(* Logix 5000 project; controller Comas_L4 vendor 1 type 14 code 193 rev 30.11; software revision 30.02; part 8 of 12 *)
(* tags used below, declared in another part *)
   AOI_Pilotage_Codeur_Vitesse_Moy : Pilotage_Vitesse_Rapide_V4;
   Axe_Codeur_Four : AXIS_CIP_DRIVE;
   Axe_Coupe_Fil : AXIS_CIP_DRIVE;
   Axe_Horizontal_Droit : AXIS_CIP_DRIVE;
   Axe_Horizontal_Gauche : AXIS_CIP_DRIVE;
   Axe_Pompe_Doseuse : AXIS_CIP_DRIVE;
   Axe_Rouleaux_Canneles : AXIS_CIP_DRIVE;
   Axe_Vertical_Droit : AXIS_CIP_DRIVE;
   Axe_Vertical_Gauche : AXIS_CIP_DRIVE;
   Axe_Virtuel_Codeur : AXIS_VIRTUAL;
   Axe_Virtuel_Maitre : AXIS_VIRTUAL;
   CamGenerator_Coupe_Fil : AOI_CamGenerator_ST;
   CamGenerator_Horizontal : AOI_CamGenerator_ST;
   CamGenerator_Vertical : AOI_CamGenerator_ST;
   CO_Acquit_defaut : BOOL;
   CO_Axe_Codeur_Four_Conv_Cons : REAL;
   CO_Axe_Codeur_Four_OK : BOOL;
   CO_Axe_Codeur_Four_PosUnwind : DINT;
   CO_Axe_Coupe_Fil_Conv_Cons : REAL;
   CO_Axe_Coupe_Fil_OK : BOOL;
   CO_Axe_Coupe_Fil_PosUnwind : DINT;
   CO_Axe_Horizontal_Droit_OK : BOOL;
   CO_Axe_Horizontal_Gauche_OK : BOOL;
   CO_Axe_Pompe_Doseuse_OK : BOOL;
   CO_Axe_Rouleaux_Canneles_OK : BOOL;
   CO_Axe_Vertical_Droit_OK : BOOL;
   CO_Axe_Vertical_Gauche_OK : BOOL;
   CO_Axe_Virtuel_Codeur_Conv_Cons : REAL;
   CO_Axe_Virtuel_Codeur_PosUnwind : DINT;
   CO_Axe_Virtuel_Maitre_Conv_Cons : REAL;
   CO_Axe_Virtuel_Maitre_PosUnwind : DINT;
   CO_BP_Coupe_Fil_Neg : BOOL;
   CO_BP_Coupe_Fil_Pos : BOOL;
   CO_BP_Horizontal_Droit_Neg : BOOL;
   CO_BP_Horizontal_Droit_Pos : BOOL;
   CO_BP_Horizontal_Gauche_Neg : BOOL;
   CO_BP_Horizontal_Gauche_Pos : BOOL;
   CO_BP_Pompe_Doseuse_Neg : BOOL;
   CO_BP_Pompe_Doseuse_Pos : BOOL;
   CO_BP_Rouleaux_Canneles_Neg : BOOL;
   CO_BP_Rouleaux_Canneles_Pos : BOOL;
   CO_BP_Vertical_Droit_Neg : BOOL;
   CO_BP_Vertical_Droit_Pos : BOOL;
   CO_BP_Vertical_Gauche_Neg : BOOL;
   CO_BP_Vertical_Gauche_Pos : BOOL;
   CO_Defaut_CamGenerator_Coupe_Fil : BOOL;
   CO_Defaut_CamGenerator_Horizontal : BOOL;
   CO_Defaut_CamGenerator_Vertical : BOOL;
   CO_Defaut_Eth_Codeur_Four : BOOL;
   CO_Defaut_Eth_Var_Coupe_Fil : BOOL;
   CO_Defaut_Eth_Var_H_Droit : BOOL;
   CO_Defaut_Eth_Var_H_Gauche : BOOL;
   CO_Defaut_Eth_Var_Pompe_Doseuse : BOOL;
   CO_Defaut_Eth_Var_Rouleaux : BOOL;
   CO_Defaut_Eth_Var_V_Droit : BOOL;
   CO_Defaut_Eth_Var_V_Gauche : BOOL;
   CO_Defaut_FDC_Amont_Horizontal_Droit : BOOL;
   CO_Defaut_FDC_Amont_Horizontal_Gauche : BOOL;
   CO_Defaut_FDC_Aval_Horizontal_Droit : BOOL;
   CO_Defaut_FDC_Aval_Horizontal_Gauche : BOOL;
   CO_Defaut_FDC_Bas_Vertical_Droit : BOOL;
   CO_Defaut_FDC_Bas_Vertical_Gauche : BOOL;
   CO_Defaut_FDC_Coupe_Fil_Droit : BOOL;
   CO_Defaut_FDC_Coupe_Fil_Gauche : BOOL;
   CO_Defaut_FDC_Haut_Vertical_Droit : BOOL;
   CO_Defaut_FDC_Haut_Vertical_Gauche : BOOL;
   CO_Defaut_Presence_Coupe_Fil : BOOL;
   CO_en_Marche : BOOL;
   CO_Machine_sans_defaut : BOOL;
   CO_Messages_En : STRING[380];
   CO_Raz_Axe : BOOL;
   CO_Temp_Vitesse_Four : REAL;
   Consigne_Acc_Decc_Manu_Degre : DINT;
   Consigne_Vitesse_Manu_Degre_Seconde : REAL;
   Consigne_Vitesse_Manu_Tour_Seconde : REAL;
   ENT_CO_Presence_Coupe_Fil : ALIAS FOR Local:2:I.Pt00.Data;
   L_Ms_Index_Codeur_Four : DINT;
   L_Ms_Index_Coupe_Fil : DINT;
   L_Ms_Index_H_Droit : DINT;
   L_Ms_Index_H_Gauche : DINT;
   L_Ms_Index_Pompe_Doseuse : DINT;
   L_Ms_Index_Rouleaux : DINT;
   L_Ms_Index_V_Droit : DINT;
   L_Ms_Index_V_Gauche : DINT;
   Message_Axe_Codeur_Four : Message_Axe;
   Message_Axe_Coupe_Fil : Message_Axe;
   Message_Axe_H_Droit : Message_Axe;
   Message_Axe_H_Gauche : Message_Axe;
   Message_Axe_Pompe_Doseuse : Message_Axe;
   Message_Axe_Rouleaux : Message_Axe;
   Message_Axe_V_Droit : Message_Axe;
   Message_Axe_V_Gauche : Message_Axe;
   Message_Defaut_Codeur_Four : STRING;
   Message_Defaut_Coupe_Fil : STRING;
   Message_Defaut_H_Droit : STRING;
   Message_Defaut_H_Gauche : STRING;
   Message_Defaut_Pompe_Doseuse : STRING;
   Message_Defaut_Rouleaux : STRING;
   Message_Defaut_V_Droit : STRING;
   Message_Defaut_V_Gauche : STRING;
   Raz_Axe_Coupe_Fil : Raz_Axe;
   Raz_Axe_H_Droit : Raz_Axe;
   Raz_Axe_H_Gauche : Raz_Axe;
   Raz_Axe_Pompe_Doseuse : Raz_Axe;
   Raz_Axe_Rouleaux : Raz_Axe;
   Raz_Axe_V_Droit : Raz_Axe;
   Raz_Axe_V_Gauche : Raz_Axe;
   RECETTE_EC : UDT_RECIPE;
   RSW_CO_Activation_Nettoyage : BOOL;
   RSW_CO_BP_Coupe_Fil_Neg : BOOL;
   RSW_CO_BP_Coupe_Fil_Pos : BOOL;
   RSW_CO_BP_Horizontal_Droit_Neg : BOOL;
   RSW_CO_BP_Horizontal_Droit_Pos : BOOL;
   RSW_CO_BP_Horizontal_Gauche_Neg : BOOL;
   RSW_CO_BP_Horizontal_Gauche_Pos : BOOL;
   RSW_CO_BP_Horizontal_Neg : BOOL;
   RSW_CO_BP_Horizontal_Pos : BOOL;
   RSW_CO_BP_Pompe_Doseuse_Neg : BOOL;
   RSW_CO_BP_Pompe_Doseuse_Pos : BOOL;
   RSW_CO_BP_Rouleaux_Canneles_Neg : BOOL;
   RSW_CO_BP_Rouleaux_Canneles_Pos : BOOL;
   RSW_CO_BP_Vertical_Droit_Neg : BOOL;
   RSW_CO_BP_Vertical_Droit_Pos : BOOL;
   RSW_CO_BP_Vertical_Gauche_Neg : BOOL;
   RSW_CO_BP_Vertical_Gauche_Pos : BOOL;
   RSW_CO_BP_Vertical_Neg : BOOL;
   RSW_CO_BP_Vertical_Pos : BOOL;
   RSW_CO_NB_Rangs_minutes : REAL;
   Test_Coupe_Fil : Test_Axe_Avec_Autorisation;
   Test_Coupe_Fil_EN : BOOL;
   Test_Horizontal_Droit : Test_Axe_Avec_Autorisation;
   Test_Horizontal_Droit_EN : BOOL;
   Test_Horizontal_Gauche : Test_Axe_Avec_Autorisation;
   Test_Horizontal_Gauche_EN : BOOL;
   Test_Pompe_Doseuse : Test_Axe_Avec_Autorisation;
   Test_Pompe_Doseuse_EN : BOOL;
   Test_Rouleaux_Canneles : Test_Axe_Avec_Autorisation;
   Test_Rouleaux_Canneles_EN : BOOL;
   Test_Vertical_Droit : Test_Axe_Avec_Autorisation;
   Test_Vertical_Droit_EN : BOOL;
   Test_Vertical_Gauche : Test_Axe_Avec_Autorisation;
   Test_Vertical_Gauche_EN : BOOL;
   Vitesse_Moy_Codeur : REAL;

PROGRAM Comas   (* main routine A00_Appel *)

ROUTINE A00_Appel   (* ladder *)
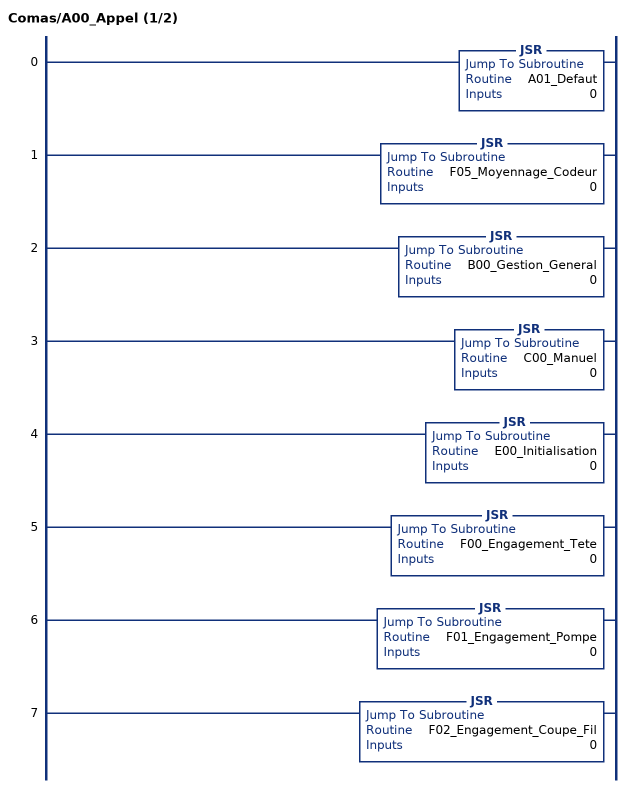
   0: JSR(A01_Defaut,0);
   1: JSR(F05_Moyennage_Codeur,0);
   2: JSR(B00_Gestion_General,0);
   3: JSR(C00_Manuel,0);
   4: JSR(E00_Initialisation,0);
   5: JSR(F00_Engagement_Tete,0);
   6: JSR(F01_Engagement_Pompe,0);
   7: JSR(F02_Engagement_Coupe_Fil,0);
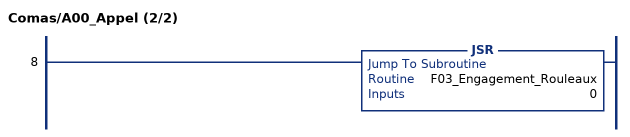
   8: JSR(F03_Engagement_Rouleaux,0);
END_ROUTINE

ROUTINE A01_Defaut   (* ladder *)
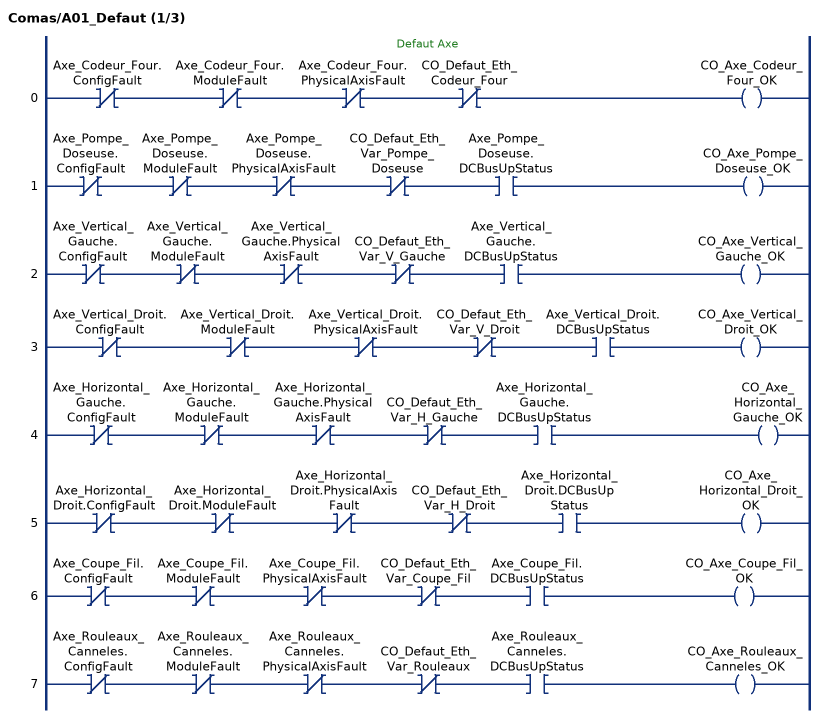
   // Defaut Axe
   0: XIO(Axe_Codeur_Four.ConfigFault)XIO(Axe_Codeur_Four.ModuleFault)XIO(Axe_Codeur_Four.PhysicalAxisFault)XIO(CO_Defaut_Eth_Codeur_Four)OTE(CO_Axe_Codeur_Four_OK);
   1: XIO(Axe_Pompe_Doseuse.ConfigFault)XIO(Axe_Pompe_Doseuse.ModuleFault)XIO(Axe_Pompe_Doseuse.PhysicalAxisFault)XIO(CO_Defaut_Eth_Var_Pompe_Doseuse)XIC(Axe_Pompe_Doseuse.DCBusUpStatus)OTE(CO_Axe_Pompe_Doseuse_OK);
   2: XIO(Axe_Vertical_Gauche.ConfigFault)XIO(Axe_Vertical_Gauche.ModuleFault)XIO(Axe_Vertical_Gauche.PhysicalAxisFault)XIO(CO_Defaut_Eth_Var_V_Gauche)XIC(Axe_Vertical_Gauche.DCBusUpStatus)OTE(CO_Axe_Vertical_Gauche_OK);
   3: XIO(Axe_Vertical_Droit.ConfigFault)XIO(Axe_Vertical_Droit.ModuleFault)XIO(Axe_Vertical_Droit.PhysicalAxisFault)XIO(CO_Defaut_Eth_Var_V_Droit)XIC(Axe_Vertical_Droit.DCBusUpStatus)OTE(CO_Axe_Vertical_Droit_OK);
   4: XIO(Axe_Horizontal_Gauche.ConfigFault)XIO(Axe_Horizontal_Gauche.ModuleFault)XIO(Axe_Horizontal_Gauche.PhysicalAxisFault)XIO(CO_Defaut_Eth_Var_H_Gauche)XIC(Axe_Horizontal_Gauche.DCBusUpStatus)OTE(CO_Axe_Horizontal_Gauche_OK);
   5: XIO(Axe_Horizontal_Droit.ConfigFault)XIO(Axe_Horizontal_Droit.ModuleFault)XIO(Axe_Horizontal_Droit.PhysicalAxisFault)XIO(CO_Defaut_Eth_Var_H_Droit)XIC(Axe_Horizontal_Droit.DCBusUpStatus)OTE(CO_Axe_Horizontal_Droit_OK);
   6: XIO(Axe_Coupe_Fil.ConfigFault)XIO(Axe_Coupe_Fil.ModuleFault)XIO(Axe_Coupe_Fil.PhysicalAxisFault)XIO(CO_Defaut_Eth_Var_Coupe_Fil)XIC(Axe_Coupe_Fil.DCBusUpStatus)OTE(CO_Axe_Coupe_Fil_OK);
   7: XIO(Axe_Rouleaux_Canneles.ConfigFault)XIO(Axe_Rouleaux_Canneles.ModuleFault)XIO(Axe_Rouleaux_Canneles.PhysicalAxisFault)XIO(CO_Defaut_Eth_Var_Rouleaux)XIC(Axe_Rouleaux_Canneles.DCBusUpStatus)OTE(CO_Axe_Rouleaux_Canneles_OK);
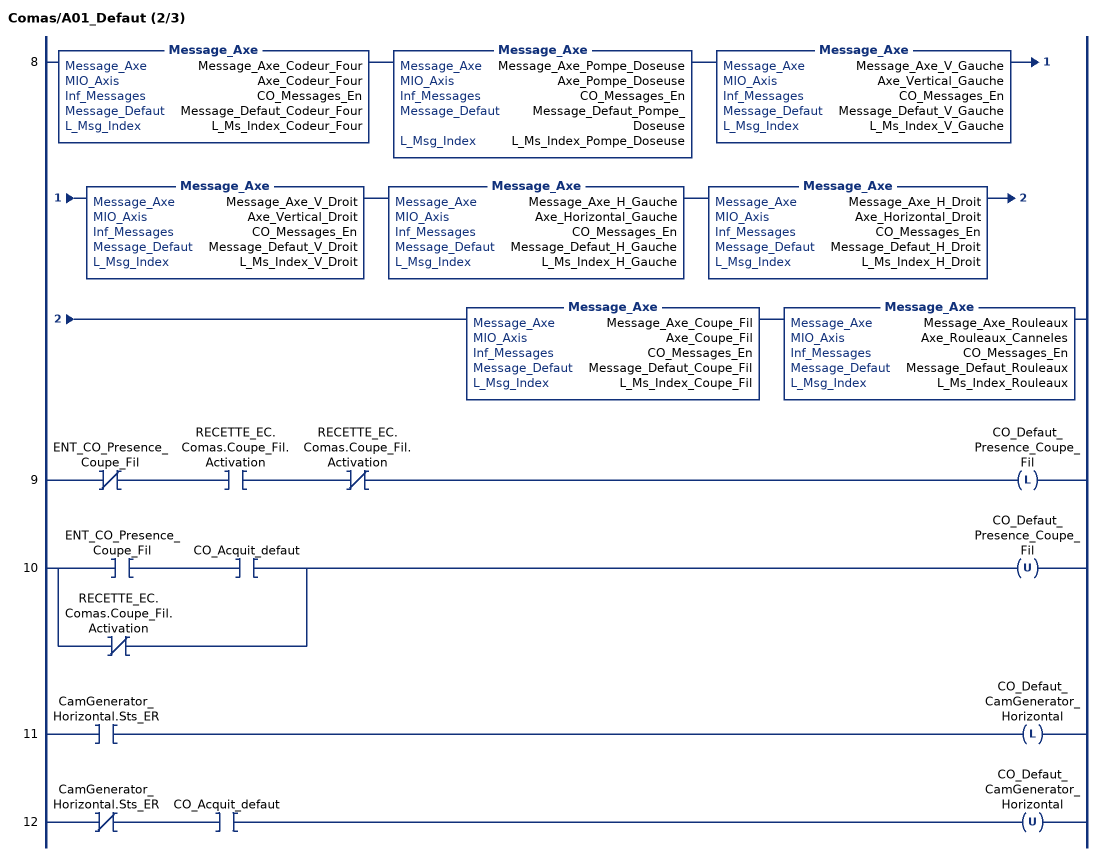
   8: Message_Axe(Message_Axe_Codeur_Four,Axe_Codeur_Four,CO_Messages_En,Message_Defaut_Codeur_Four,L_Ms_Index_Codeur_Four)Message_Axe(Message_Axe_Pompe_Doseuse,Axe_Pompe_Doseuse,CO_Messages_En,Message_Defaut_Pompe_Doseuse,L_Ms_Index_Pompe_Doseuse)Message_Axe(Message_Axe_V_Gauche,Axe_Vertical_Gauche,CO_Messages_En,Message_Defaut_V_Gauche,L_Ms_Index_V_Gauche)Message_Axe(Message_Axe_V_Droit,Axe_Vertical_Droit,CO_Messages_En,Message_Defaut_V_Droit,L_Ms_Index_V_Droit)Message_Axe(Message_Axe_H_Gauche,Axe_Horizontal_Gauche,CO_Messages_En,Message_Defaut_H_Gauche,L_Ms_Index_H_Gauche)Message_Axe(Message_Axe_H_Droit,Axe_Horizontal_Droit,CO_Messages_En,Message_Defaut_H_Droit,L_Ms_Index_H_Droit)Message_Axe(Message_Axe_Coupe_Fil,Axe_Coupe_Fil,CO_Messages_En,Message_Defaut_Coupe_Fil,L_Ms_Index_Coupe_Fil)Message_Axe(Message_Axe_Rouleaux,Axe_Rouleaux_Canneles,CO_Messages_En,Message_Defaut_Rouleaux,L_Ms_Index_Rouleaux);
   9: XIO(ENT_CO_Presence_Coupe_Fil)XIC(RECETTE_EC.Comas.Coupe_Fil.Activation)XIO(RECETTE_EC.Comas.Coupe_Fil.Activation)OTL(CO_Defaut_Presence_Coupe_Fil);
   10: [XIC(ENT_CO_Presence_Coupe_Fil) XIC(CO_Acquit_defaut) ,XIO(RECETTE_EC.Comas.Coupe_Fil.Activation) ]OTU(CO_Defaut_Presence_Coupe_Fil);
   11: XIC(CamGenerator_Horizontal.Sts_ER)OTL(CO_Defaut_CamGenerator_Horizontal);
   12: XIO(CamGenerator_Horizontal.Sts_ER)XIC(CO_Acquit_defaut)OTU(CO_Defaut_CamGenerator_Horizontal);
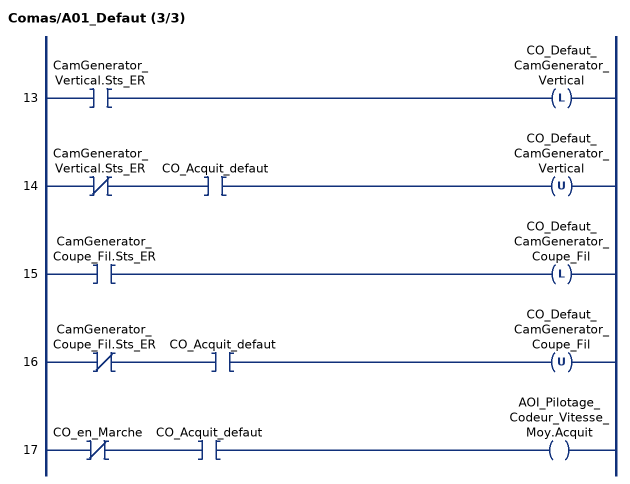
   13: XIC(CamGenerator_Vertical.Sts_ER)OTL(CO_Defaut_CamGenerator_Vertical);
   14: XIO(CamGenerator_Vertical.Sts_ER)XIC(CO_Acquit_defaut)OTU(CO_Defaut_CamGenerator_Vertical);
   15: XIC(CamGenerator_Coupe_Fil.Sts_ER)OTL(CO_Defaut_CamGenerator_Coupe_Fil);
   16: XIO(CamGenerator_Coupe_Fil.Sts_ER)XIC(CO_Acquit_defaut)OTU(CO_Defaut_CamGenerator_Coupe_Fil);
   17: XIO(CO_en_Marche)XIC(CO_Acquit_defaut)OTE(AOI_Pilotage_Codeur_Vitesse_Moy.Acquit);
END_ROUTINE

ROUTINE B00_Gestion_General   (* ladder *)
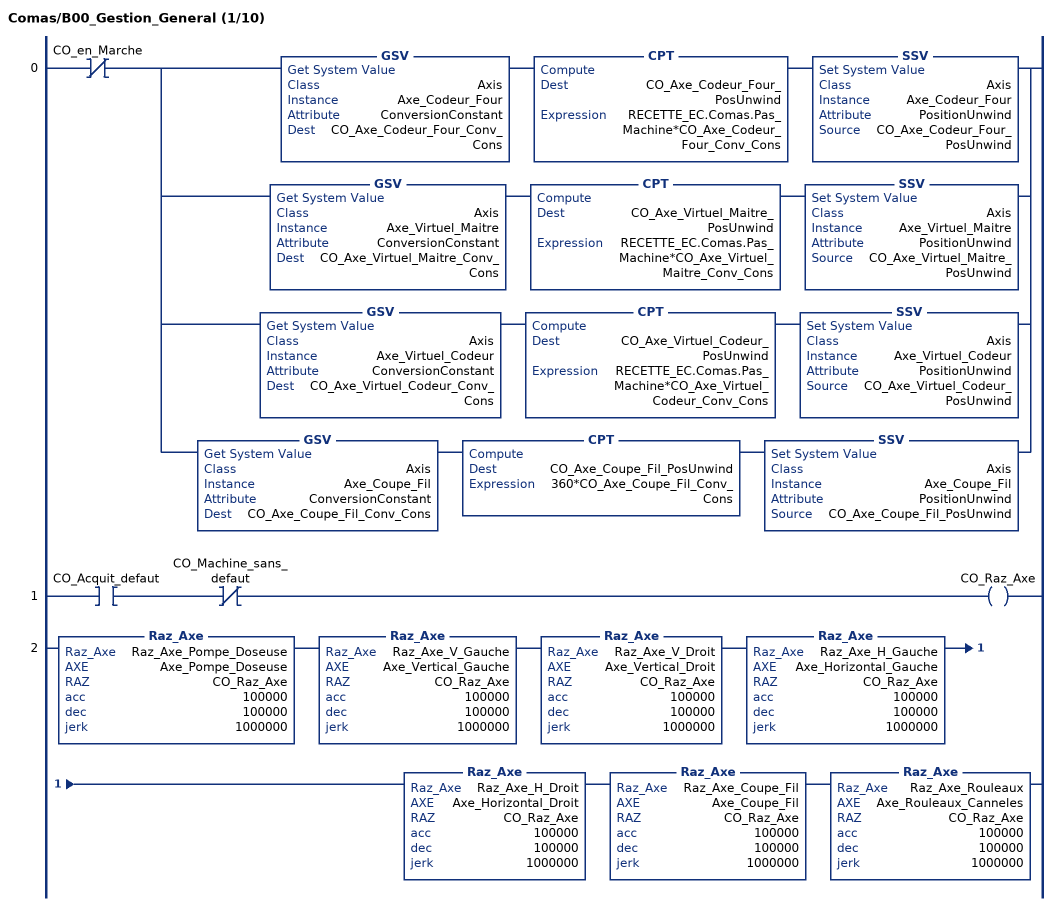
   0: XIO(CO_en_Marche)[GSV(Axis,Axe_Codeur_Four,ConversionConstant,CO_Axe_Codeur_Four_Conv_Cons) CPT(CO_Axe_Codeur_Four_PosUnwind,RECETTE_EC.Comas.Pas_Machine*CO_Axe_Codeur_Four_Conv_Cons) SSV(Axis,Axe_Codeur_Four,PositionUnwind,CO_Axe_Codeur_Four_PosUnwind) ,GSV(Axis,Axe_Virtuel_Maitre,ConversionConstant,CO_Axe_Virtuel_Maitre_Conv_Cons) CPT(CO_Axe_Virtuel_Maitre_PosUnwind,RECETTE_EC.Comas.Pas_Machine*CO_Axe_Virtuel_Maitre_Conv_Cons) SSV(Axis,Axe_Virtuel_Maitre,PositionUnwind,CO_Axe_Virtuel_Maitre_PosUnwind) ,GSV(Axis,Axe_Virtuel_Codeur,ConversionConstant,CO_Axe_Virtuel_Codeur_Conv_Cons) CPT(CO_Axe_Virtuel_Codeur_PosUnwind,RECETTE_EC.Comas.Pas_Machine*CO_Axe_Virtuel_Codeur_Conv_Cons) SSV(Axis,Axe_Virtuel_Codeur,PositionUnwind,CO_Axe_Virtuel_Codeur_PosUnwind) ,GSV(Axis,Axe_Coupe_Fil,ConversionConstant,CO_Axe_Coupe_Fil_Conv_Cons) CPT(CO_Axe_Coupe_Fil_PosUnwind,360*CO_Axe_Coupe_Fil_Conv_Cons) SSV(Axis,Axe_Coupe_Fil,PositionUnwind,CO_Axe_Coupe_Fil_PosUnwind) ];
   1: XIC(CO_Acquit_defaut)XIO(CO_Machine_sans_defaut)OTE(CO_Raz_Axe);
   2: Raz_Axe(Raz_Axe_Pompe_Doseuse,Axe_Pompe_Doseuse,CO_Raz_Axe,100000,100000,1000000)Raz_Axe(Raz_Axe_V_Gauche,Axe_Vertical_Gauche,CO_Raz_Axe,100000,100000,1000000)Raz_Axe(Raz_Axe_V_Droit,Axe_Vertical_Droit,CO_Raz_Axe,100000,100000,1000000)Raz_Axe(Raz_Axe_H_Gauche,Axe_Horizontal_Gauche,CO_Raz_Axe,100000,100000,1000000)Raz_Axe(Raz_Axe_H_Droit,Axe_Horizontal_Droit,CO_Raz_Axe,100000,100000,1000000)Raz_Axe(Raz_Axe_Coupe_Fil,Axe_Coupe_Fil,CO_Raz_Axe,100000,100000,1000000)Raz_Axe(Raz_Axe_Rouleaux,Axe_Rouleaux_Canneles,CO_Raz_Axe,100000,100000,1000000);
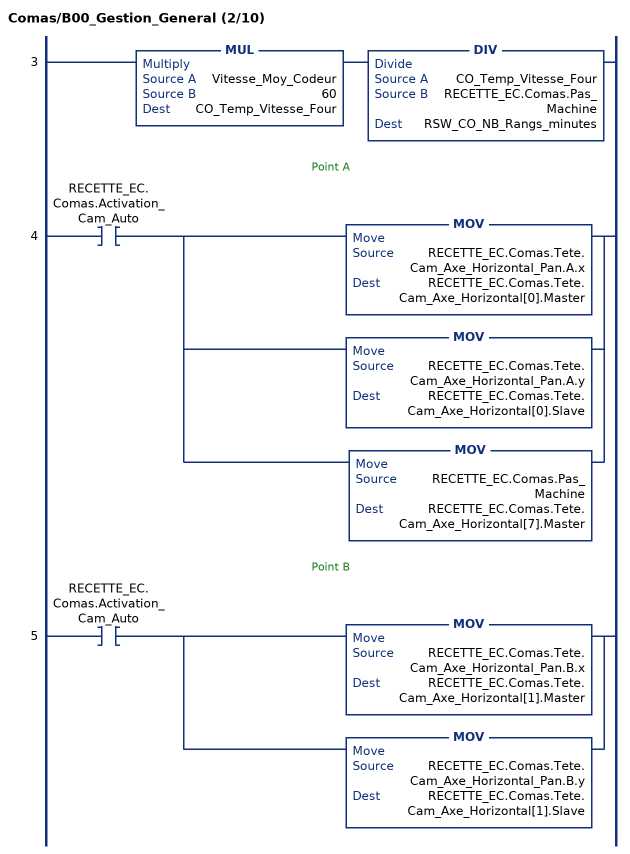
   3: MUL(Vitesse_Moy_Codeur,60,CO_Temp_Vitesse_Four)DIV(CO_Temp_Vitesse_Four,RECETTE_EC.Comas.Pas_Machine,RSW_CO_NB_Rangs_minutes);
   // Point A
   4: XIC(RECETTE_EC.Comas.Activation_Cam_Auto)[MOV(RECETTE_EC.Comas.Tete.Cam_Axe_Horizontal_Pan.A.x,RECETTE_EC.Comas.Tete.Cam_Axe_Horizontal[0].Master) ,MOV(RECETTE_EC.Comas.Tete.Cam_Axe_Horizontal_Pan.A.y,RECETTE_EC.Comas.Tete.Cam_Axe_Horizontal[0].Slave) ,MOV(RECETTE_EC.Comas.Pas_Machine,RECETTE_EC.Comas.Tete.Cam_Axe_Horizontal[7].Master) ];
   // Point B
   5: XIC(RECETTE_EC.Comas.Activation_Cam_Auto)[MOV(RECETTE_EC.Comas.Tete.Cam_Axe_Horizontal_Pan.B.x,RECETTE_EC.Comas.Tete.Cam_Axe_Horizontal[1].Master) ,MOV(RECETTE_EC.Comas.Tete.Cam_Axe_Horizontal_Pan.B.y,RECETTE_EC.Comas.Tete.Cam_Axe_Horizontal[1].Slave) ];
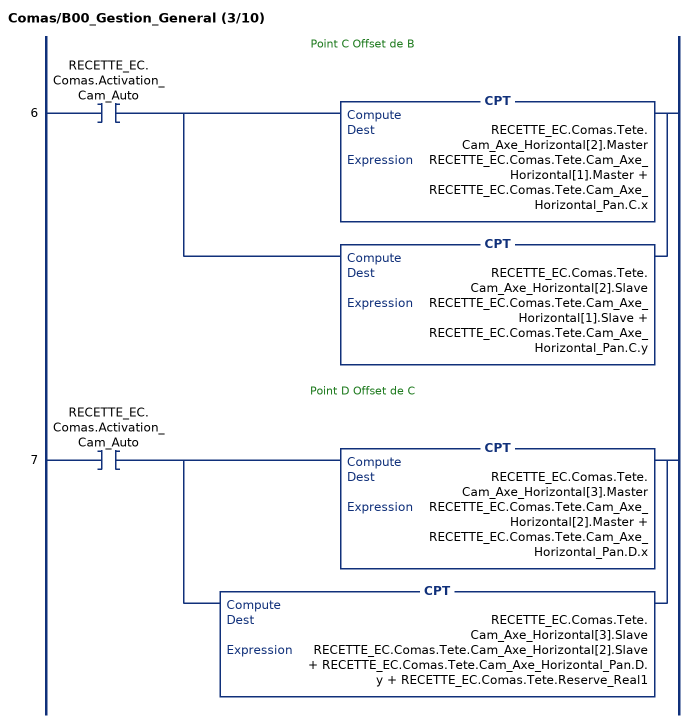
   // Point C Offset de B
   6: XIC(RECETTE_EC.Comas.Activation_Cam_Auto)[CPT(RECETTE_EC.Comas.Tete.Cam_Axe_Horizontal[2].Master,RECETTE_EC.Comas.Tete.Cam_Axe_Horizontal[1].Master + RECETTE_EC.Comas.Tete.Cam_Axe_Horizontal_Pan.C.x) ,CPT(RECETTE_EC.Comas.Tete.Cam_Axe_Horizontal[2].Slave,RECETTE_EC.Comas.Tete.Cam_Axe_Horizontal[1].Slave + RECETTE_EC.Comas.Tete.Cam_Axe_Horizontal_Pan.C.y) ];
   // Point D Offset de C
   7: XIC(RECETTE_EC.Comas.Activation_Cam_Auto)[CPT(RECETTE_EC.Comas.Tete.Cam_Axe_Horizontal[3].Master,RECETTE_EC.Comas.Tete.Cam_Axe_Horizontal[2].Master + RECETTE_EC.Comas.Tete.Cam_Axe_Horizontal_Pan.D.x) ,CPT(RECETTE_EC.Comas.Tete.Cam_Axe_Horizontal[3].Slave,RECETTE_EC.Comas.Tete.Cam_Axe_Horizontal[2].Slave + RECETTE_EC.Comas.Tete.Cam_Axe_Horizontal_Pan.D.y + RECETTE_EC.Comas.Tete.Reserve_Real1) ];
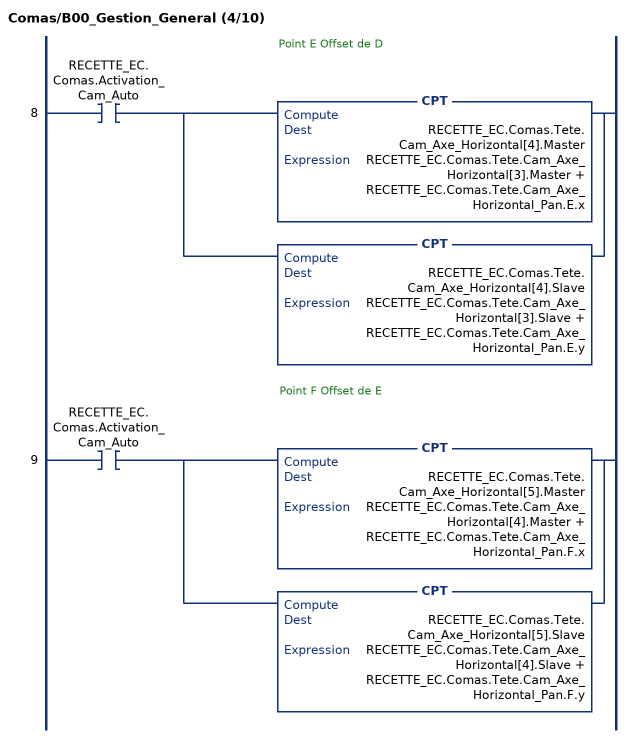
   // Point E Offset de D
   8: XIC(RECETTE_EC.Comas.Activation_Cam_Auto)[CPT(RECETTE_EC.Comas.Tete.Cam_Axe_Horizontal[4].Master,RECETTE_EC.Comas.Tete.Cam_Axe_Horizontal[3].Master + RECETTE_EC.Comas.Tete.Cam_Axe_Horizontal_Pan.E.x) ,CPT(RECETTE_EC.Comas.Tete.Cam_Axe_Horizontal[4].Slave,RECETTE_EC.Comas.Tete.Cam_Axe_Horizontal[3].Slave + RECETTE_EC.Comas.Tete.Cam_Axe_Horizontal_Pan.E.y) ];
   // Point F Offset de E
   9: XIC(RECETTE_EC.Comas.Activation_Cam_Auto)[CPT(RECETTE_EC.Comas.Tete.Cam_Axe_Horizontal[5].Master,RECETTE_EC.Comas.Tete.Cam_Axe_Horizontal[4].Master + RECETTE_EC.Comas.Tete.Cam_Axe_Horizontal_Pan.F.x) ,CPT(RECETTE_EC.Comas.Tete.Cam_Axe_Horizontal[5].Slave,RECETTE_EC.Comas.Tete.Cam_Axe_Horizontal[4].Slave + RECETTE_EC.Comas.Tete.Cam_Axe_Horizontal_Pan.F.y) ];
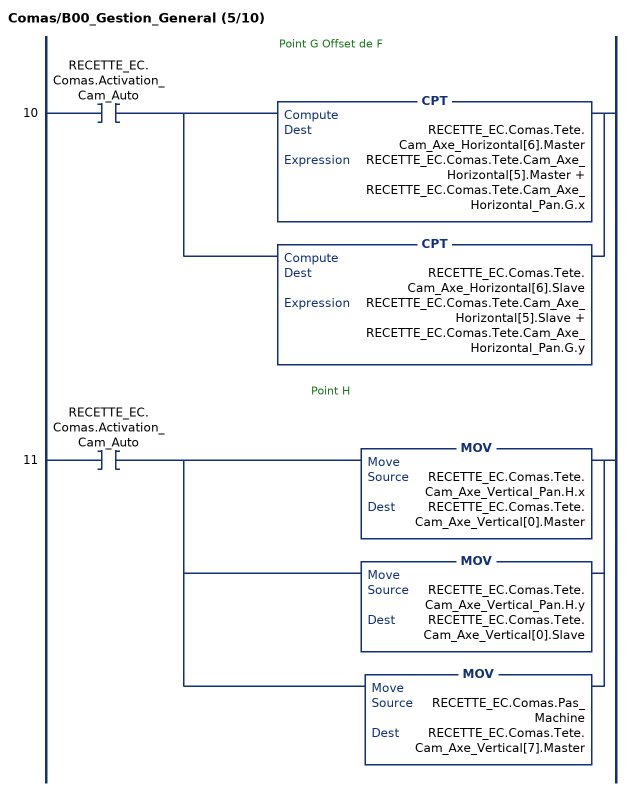
   // Point G Offset de F
   10: XIC(RECETTE_EC.Comas.Activation_Cam_Auto)[CPT(RECETTE_EC.Comas.Tete.Cam_Axe_Horizontal[6].Master,RECETTE_EC.Comas.Tete.Cam_Axe_Horizontal[5].Master + RECETTE_EC.Comas.Tete.Cam_Axe_Horizontal_Pan.G.x) ,CPT(RECETTE_EC.Comas.Tete.Cam_Axe_Horizontal[6].Slave,RECETTE_EC.Comas.Tete.Cam_Axe_Horizontal[5].Slave + RECETTE_EC.Comas.Tete.Cam_Axe_Horizontal_Pan.G.y) ];
   // Point H
   11: XIC(RECETTE_EC.Comas.Activation_Cam_Auto)[MOV(RECETTE_EC.Comas.Tete.Cam_Axe_Vertical_Pan.H.x,RECETTE_EC.Comas.Tete.Cam_Axe_Vertical[0].Master) ,MOV(RECETTE_EC.Comas.Tete.Cam_Axe_Vertical_Pan.H.y,RECETTE_EC.Comas.Tete.Cam_Axe_Vertical[0].Slave) ,MOV(RECETTE_EC.Comas.Pas_Machine,RECETTE_EC.Comas.Tete.Cam_Axe_Vertical[7].Master) ];
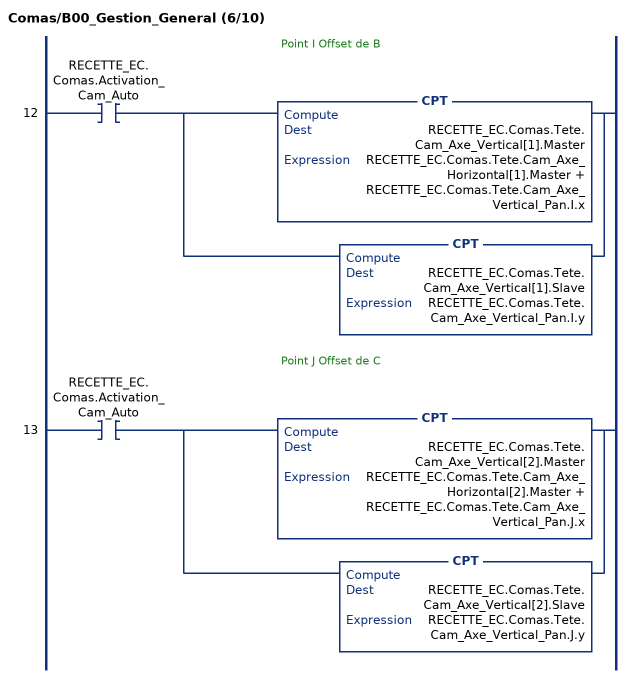
   // Point I Offset de B
   12: XIC(RECETTE_EC.Comas.Activation_Cam_Auto)[CPT(RECETTE_EC.Comas.Tete.Cam_Axe_Vertical[1].Master,RECETTE_EC.Comas.Tete.Cam_Axe_Horizontal[1].Master + RECETTE_EC.Comas.Tete.Cam_Axe_Vertical_Pan.I.x) ,CPT(RECETTE_EC.Comas.Tete.Cam_Axe_Vertical[1].Slave,RECETTE_EC.Comas.Tete.Cam_Axe_Vertical_Pan.I.y) ];
   // Point J Offset de C
   13: XIC(RECETTE_EC.Comas.Activation_Cam_Auto)[CPT(RECETTE_EC.Comas.Tete.Cam_Axe_Vertical[2].Master,RECETTE_EC.Comas.Tete.Cam_Axe_Horizontal[2].Master + RECETTE_EC.Comas.Tete.Cam_Axe_Vertical_Pan.J.x) ,CPT(RECETTE_EC.Comas.Tete.Cam_Axe_Vertical[2].Slave,RECETTE_EC.Comas.Tete.Cam_Axe_Vertical_Pan.J.y) ];
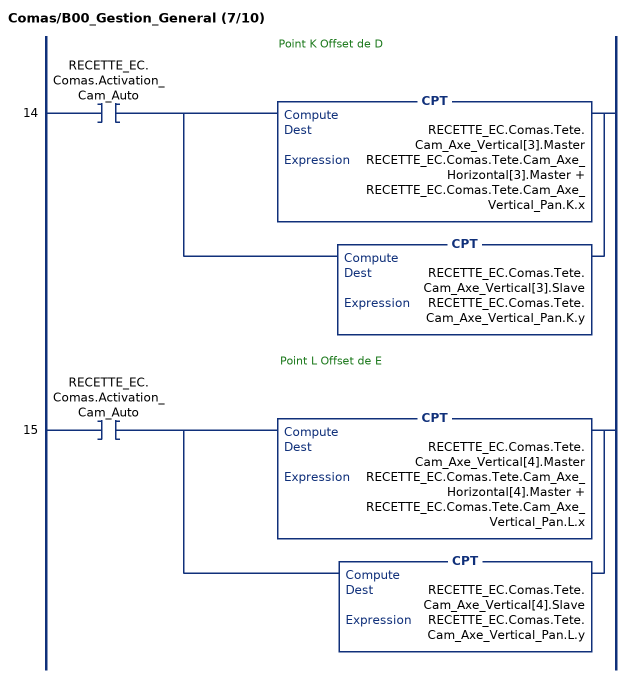
   // Point K Offset de D
   14: XIC(RECETTE_EC.Comas.Activation_Cam_Auto)[CPT(RECETTE_EC.Comas.Tete.Cam_Axe_Vertical[3].Master,RECETTE_EC.Comas.Tete.Cam_Axe_Horizontal[3].Master + RECETTE_EC.Comas.Tete.Cam_Axe_Vertical_Pan.K.x) ,CPT(RECETTE_EC.Comas.Tete.Cam_Axe_Vertical[3].Slave,RECETTE_EC.Comas.Tete.Cam_Axe_Vertical_Pan.K.y) ];
   // Point L Offset de E
   15: XIC(RECETTE_EC.Comas.Activation_Cam_Auto)[CPT(RECETTE_EC.Comas.Tete.Cam_Axe_Vertical[4].Master,RECETTE_EC.Comas.Tete.Cam_Axe_Horizontal[4].Master + RECETTE_EC.Comas.Tete.Cam_Axe_Vertical_Pan.L.x) ,CPT(RECETTE_EC.Comas.Tete.Cam_Axe_Vertical[4].Slave,RECETTE_EC.Comas.Tete.Cam_Axe_Vertical_Pan.L.y) ];
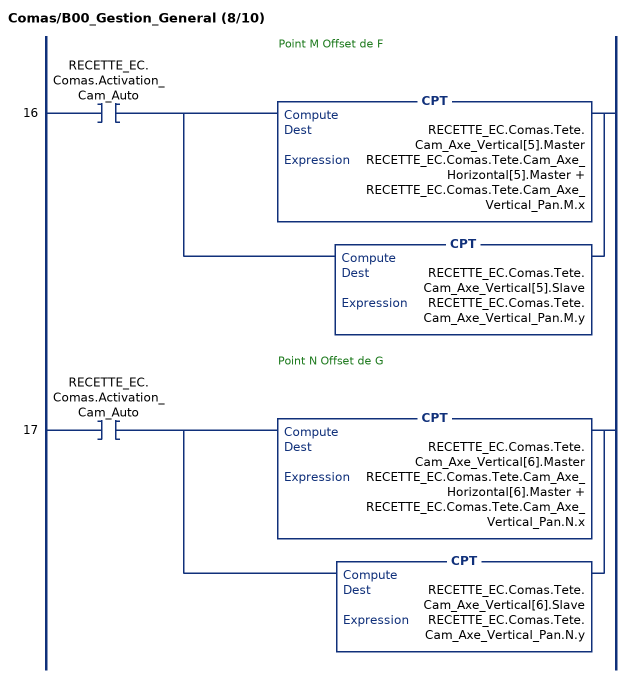
   // Point M Offset de F
   16: XIC(RECETTE_EC.Comas.Activation_Cam_Auto)[CPT(RECETTE_EC.Comas.Tete.Cam_Axe_Vertical[5].Master,RECETTE_EC.Comas.Tete.Cam_Axe_Horizontal[5].Master + RECETTE_EC.Comas.Tete.Cam_Axe_Vertical_Pan.M.x) ,CPT(RECETTE_EC.Comas.Tete.Cam_Axe_Vertical[5].Slave,RECETTE_EC.Comas.Tete.Cam_Axe_Vertical_Pan.M.y) ];
   // Point N Offset de G
   17: XIC(RECETTE_EC.Comas.Activation_Cam_Auto)[CPT(RECETTE_EC.Comas.Tete.Cam_Axe_Vertical[6].Master,RECETTE_EC.Comas.Tete.Cam_Axe_Horizontal[6].Master + RECETTE_EC.Comas.Tete.Cam_Axe_Vertical_Pan.N.x) ,CPT(RECETTE_EC.Comas.Tete.Cam_Axe_Vertical[6].Slave,RECETTE_EC.Comas.Tete.Cam_Axe_Vertical_Pan.N.y) ];
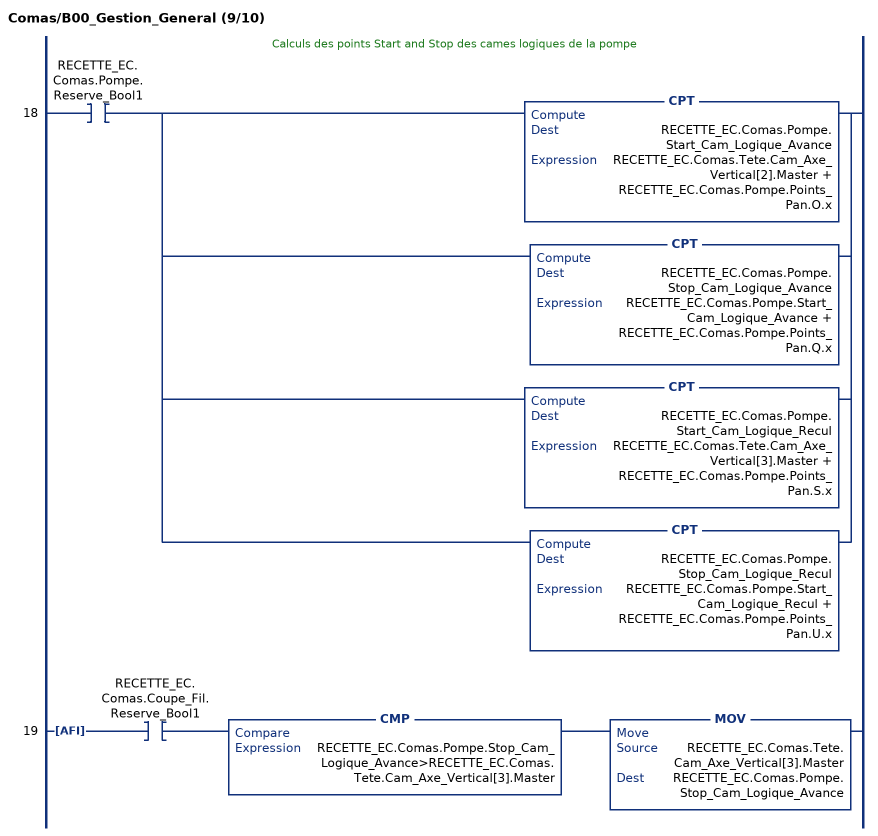
   // Calculs des points Start and Stop des cames logiques de la pompe
   18: XIC(RECETTE_EC.Comas.Pompe.Reserve_Bool1)[CPT(RECETTE_EC.Comas.Pompe.Start_Cam_Logique_Avance,RECETTE_EC.Comas.Tete.Cam_Axe_Vertical[2].Master + RECETTE_EC.Comas.Pompe.Points_Pan.O.x) ,CPT(RECETTE_EC.Comas.Pompe.Stop_Cam_Logique_Avance,RECETTE_EC.Comas.Pompe.Start_Cam_Logique_Avance + RECETTE_EC.Comas.Pompe.Points_Pan.Q.x) ,CPT(RECETTE_EC.Comas.Pompe.Start_Cam_Logique_Recul,RECETTE_EC.Comas.Tete.Cam_Axe_Vertical[3].Master + RECETTE_EC.Comas.Pompe.Points_Pan.S.x) ,CPT(RECETTE_EC.Comas.Pompe.Stop_Cam_Logique_Recul,RECETTE_EC.Comas.Pompe.Start_Cam_Logique_Recul + RECETTE_EC.Comas.Pompe.Points_Pan.U.x) ];
   19: AFI()XIC(RECETTE_EC.Comas.Coupe_Fil.Reserve_Bool1)CMP(RECETTE_EC.Comas.Pompe.Stop_Cam_Logique_Avance>RECETTE_EC.Comas.Tete.Cam_Axe_Vertical[3].Master)MOV(RECETTE_EC.Comas.Tete.Cam_Axe_Vertical[3].Master,RECETTE_EC.Comas.Pompe.Stop_Cam_Logique_Avance);
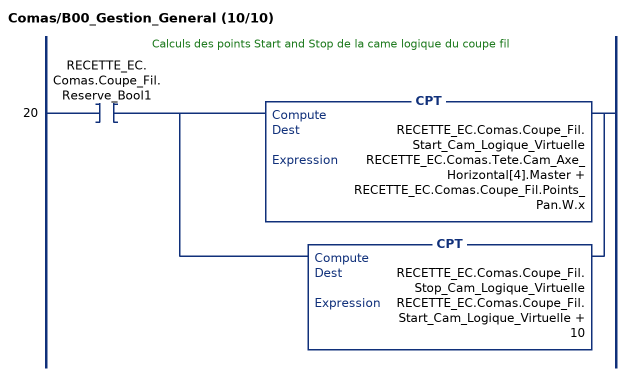
   // Calculs des points Start and Stop de la came logique du coupe fil
   20: XIC(RECETTE_EC.Comas.Coupe_Fil.Reserve_Bool1)[CPT(RECETTE_EC.Comas.Coupe_Fil.Start_Cam_Logique_Virtuelle,RECETTE_EC.Comas.Tete.Cam_Axe_Horizontal[4].Master + RECETTE_EC.Comas.Coupe_Fil.Points_Pan.W.x) ,CPT(RECETTE_EC.Comas.Coupe_Fil.Stop_Cam_Logique_Virtuelle,RECETTE_EC.Comas.Coupe_Fil.Start_Cam_Logique_Virtuelle + 10) ];
END_ROUTINE

ROUTINE C00_Manuel   (* ladder *)
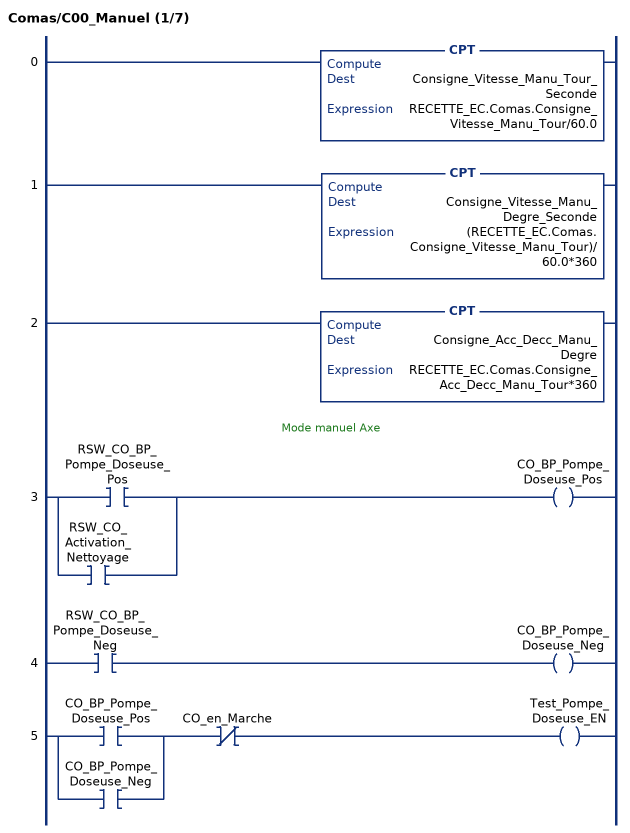
   0: CPT(Consigne_Vitesse_Manu_Tour_Seconde,RECETTE_EC.Comas.Consigne_Vitesse_Manu_Tour/60.0);
   1: CPT(Consigne_Vitesse_Manu_Degre_Seconde,(RECETTE_EC.Comas.Consigne_Vitesse_Manu_Tour)/60.0*360);
   2: CPT(Consigne_Acc_Decc_Manu_Degre,RECETTE_EC.Comas.Consigne_Acc_Decc_Manu_Tour*360);
   // Mode manuel Axe
   3: [XIC(RSW_CO_BP_Pompe_Doseuse_Pos) ,XIC(RSW_CO_Activation_Nettoyage) ]OTE(CO_BP_Pompe_Doseuse_Pos);
   4: XIC(RSW_CO_BP_Pompe_Doseuse_Neg)OTE(CO_BP_Pompe_Doseuse_Neg);
   5: [XIC(CO_BP_Pompe_Doseuse_Pos) ,XIC(CO_BP_Pompe_Doseuse_Neg) ]XIO(CO_en_Marche)OTE(Test_Pompe_Doseuse_EN);
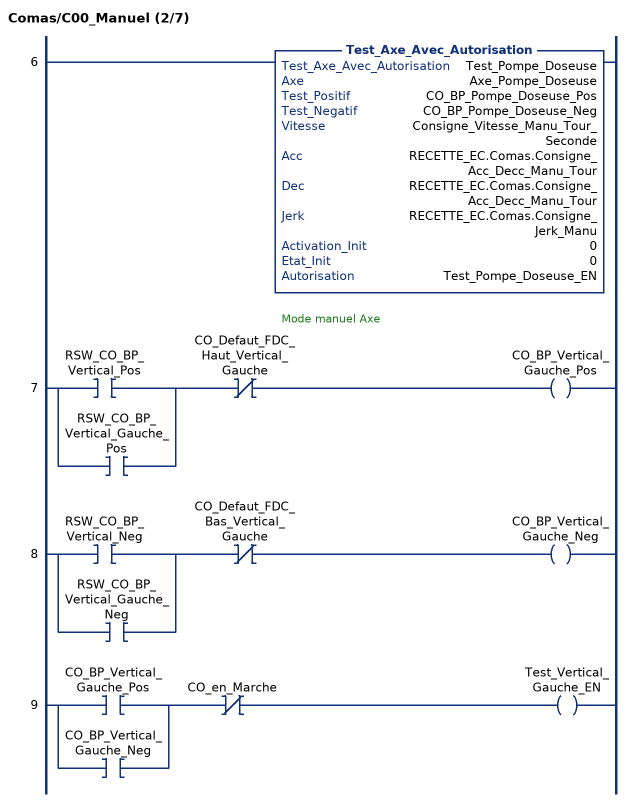
   6: Test_Axe_Avec_Autorisation(Test_Pompe_Doseuse,Axe_Pompe_Doseuse,CO_BP_Pompe_Doseuse_Pos,CO_BP_Pompe_Doseuse_Neg,Consigne_Vitesse_Manu_Tour_Seconde,RECETTE_EC.Comas.Consigne_Acc_Decc_Manu_Tour,RECETTE_EC.Comas.Consigne_Acc_Decc_Manu_Tour,RECETTE_EC.Comas.Consigne_Jerk_Manu,0,0,Test_Pompe_Doseuse_EN);
   // Mode manuel Axe
   7: [XIC(RSW_CO_BP_Vertical_Pos) ,XIC(RSW_CO_BP_Vertical_Gauche_Pos) ]XIO(CO_Defaut_FDC_Haut_Vertical_Gauche)OTE(CO_BP_Vertical_Gauche_Pos);
   8: [XIC(RSW_CO_BP_Vertical_Neg) ,XIC(RSW_CO_BP_Vertical_Gauche_Neg) ]XIO(CO_Defaut_FDC_Bas_Vertical_Gauche)OTE(CO_BP_Vertical_Gauche_Neg);
   9: [XIC(CO_BP_Vertical_Gauche_Pos) ,XIC(CO_BP_Vertical_Gauche_Neg) ]XIO(CO_en_Marche)OTE(Test_Vertical_Gauche_EN);
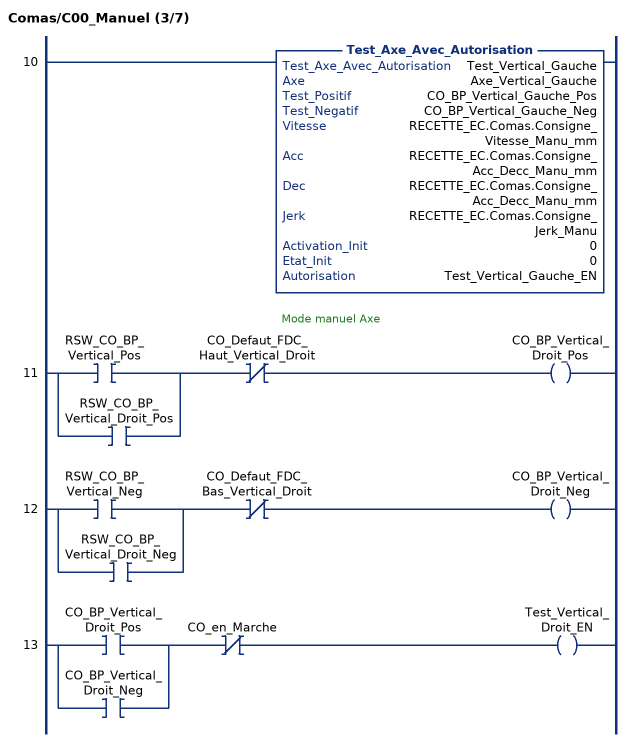
   10: Test_Axe_Avec_Autorisation(Test_Vertical_Gauche,Axe_Vertical_Gauche,CO_BP_Vertical_Gauche_Pos,CO_BP_Vertical_Gauche_Neg,RECETTE_EC.Comas.Consigne_Vitesse_Manu_mm,RECETTE_EC.Comas.Consigne_Acc_Decc_Manu_mm,RECETTE_EC.Comas.Consigne_Acc_Decc_Manu_mm,RECETTE_EC.Comas.Consigne_Jerk_Manu,0,0,Test_Vertical_Gauche_EN);
   // Mode manuel Axe
   11: [XIC(RSW_CO_BP_Vertical_Pos) ,XIC(RSW_CO_BP_Vertical_Droit_Pos) ]XIO(CO_Defaut_FDC_Haut_Vertical_Droit)OTE(CO_BP_Vertical_Droit_Pos);
   12: [XIC(RSW_CO_BP_Vertical_Neg) ,XIC(RSW_CO_BP_Vertical_Droit_Neg) ]XIO(CO_Defaut_FDC_Bas_Vertical_Droit)OTE(CO_BP_Vertical_Droit_Neg);
   13: [XIC(CO_BP_Vertical_Droit_Pos) ,XIC(CO_BP_Vertical_Droit_Neg) ]XIO(CO_en_Marche)OTE(Test_Vertical_Droit_EN);
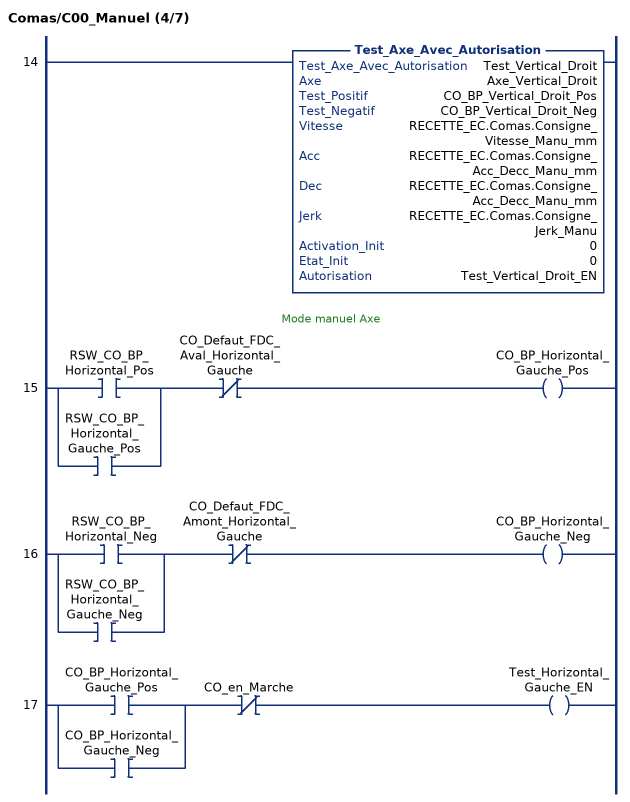
   14: Test_Axe_Avec_Autorisation(Test_Vertical_Droit,Axe_Vertical_Droit,CO_BP_Vertical_Droit_Pos,CO_BP_Vertical_Droit_Neg,RECETTE_EC.Comas.Consigne_Vitesse_Manu_mm,RECETTE_EC.Comas.Consigne_Acc_Decc_Manu_mm,RECETTE_EC.Comas.Consigne_Acc_Decc_Manu_mm,RECETTE_EC.Comas.Consigne_Jerk_Manu,0,0,Test_Vertical_Droit_EN);
   // Mode manuel Axe
   15: [XIC(RSW_CO_BP_Horizontal_Pos) ,XIC(RSW_CO_BP_Horizontal_Gauche_Pos) ]XIO(CO_Defaut_FDC_Aval_Horizontal_Gauche)OTE(CO_BP_Horizontal_Gauche_Pos);
   16: [XIC(RSW_CO_BP_Horizontal_Neg) ,XIC(RSW_CO_BP_Horizontal_Gauche_Neg) ]XIO(CO_Defaut_FDC_Amont_Horizontal_Gauche)OTE(CO_BP_Horizontal_Gauche_Neg);
   17: [XIC(CO_BP_Horizontal_Gauche_Pos) ,XIC(CO_BP_Horizontal_Gauche_Neg) ]XIO(CO_en_Marche)OTE(Test_Horizontal_Gauche_EN);
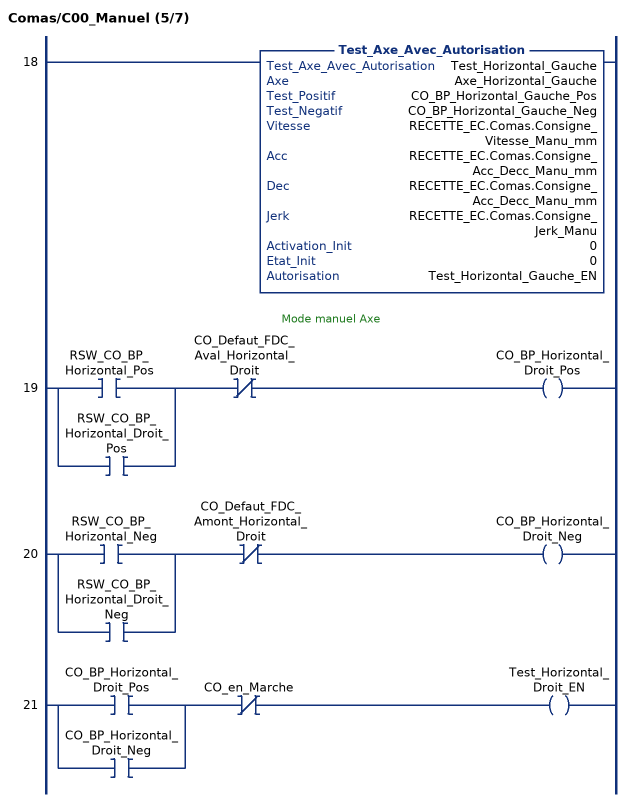
   18: Test_Axe_Avec_Autorisation(Test_Horizontal_Gauche,Axe_Horizontal_Gauche,CO_BP_Horizontal_Gauche_Pos,CO_BP_Horizontal_Gauche_Neg,RECETTE_EC.Comas.Consigne_Vitesse_Manu_mm,RECETTE_EC.Comas.Consigne_Acc_Decc_Manu_mm,RECETTE_EC.Comas.Consigne_Acc_Decc_Manu_mm,RECETTE_EC.Comas.Consigne_Jerk_Manu,0,0,Test_Horizontal_Gauche_EN);
   // Mode manuel Axe
   19: [XIC(RSW_CO_BP_Horizontal_Pos) ,XIC(RSW_CO_BP_Horizontal_Droit_Pos) ]XIO(CO_Defaut_FDC_Aval_Horizontal_Droit)OTE(CO_BP_Horizontal_Droit_Pos);
   20: [XIC(RSW_CO_BP_Horizontal_Neg) ,XIC(RSW_CO_BP_Horizontal_Droit_Neg) ]XIO(CO_Defaut_FDC_Amont_Horizontal_Droit)OTE(CO_BP_Horizontal_Droit_Neg);
   21: [XIC(CO_BP_Horizontal_Droit_Pos) ,XIC(CO_BP_Horizontal_Droit_Neg) ]XIO(CO_en_Marche)OTE(Test_Horizontal_Droit_EN);
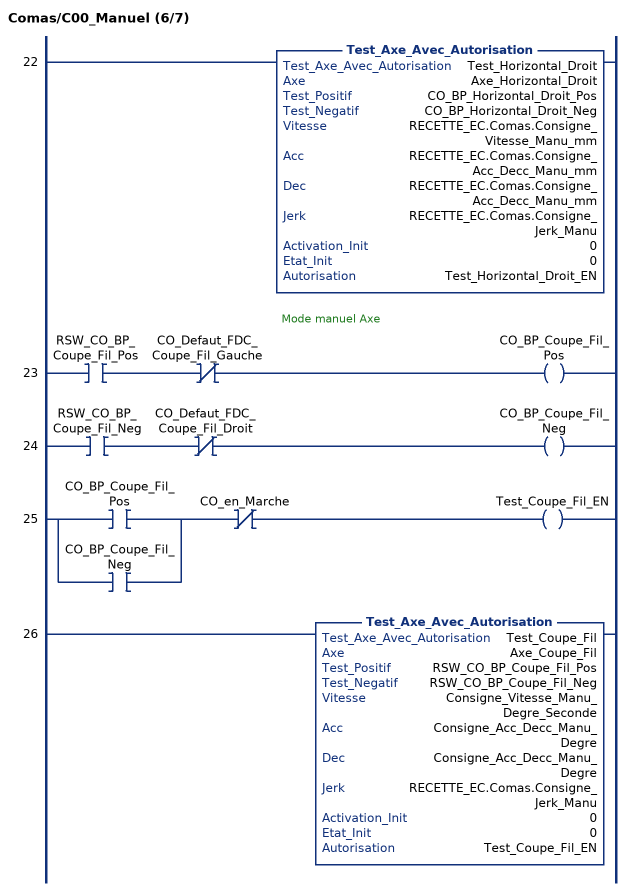
   22: Test_Axe_Avec_Autorisation(Test_Horizontal_Droit,Axe_Horizontal_Droit,CO_BP_Horizontal_Droit_Pos,CO_BP_Horizontal_Droit_Neg,RECETTE_EC.Comas.Consigne_Vitesse_Manu_mm,RECETTE_EC.Comas.Consigne_Acc_Decc_Manu_mm,RECETTE_EC.Comas.Consigne_Acc_Decc_Manu_mm,RECETTE_EC.Comas.Consigne_Jerk_Manu,0,0,Test_Horizontal_Droit_EN);
   // Mode manuel Axe
   23: XIC(RSW_CO_BP_Coupe_Fil_Pos)XIO(CO_Defaut_FDC_Coupe_Fil_Gauche)OTE(CO_BP_Coupe_Fil_Pos);
   24: XIC(RSW_CO_BP_Coupe_Fil_Neg)XIO(CO_Defaut_FDC_Coupe_Fil_Droit)OTE(CO_BP_Coupe_Fil_Neg);
   25: [XIC(CO_BP_Coupe_Fil_Pos) ,XIC(CO_BP_Coupe_Fil_Neg) ]XIO(CO_en_Marche)OTE(Test_Coupe_Fil_EN);
   26: Test_Axe_Avec_Autorisation(Test_Coupe_Fil,Axe_Coupe_Fil,RSW_CO_BP_Coupe_Fil_Pos,RSW_CO_BP_Coupe_Fil_Neg,Consigne_Vitesse_Manu_Degre_Seconde,Consigne_Acc_Decc_Manu_Degre,Consigne_Acc_Decc_Manu_Degre,RECETTE_EC.Comas.Consigne_Jerk_Manu,0,0,Test_Coupe_Fil_EN);
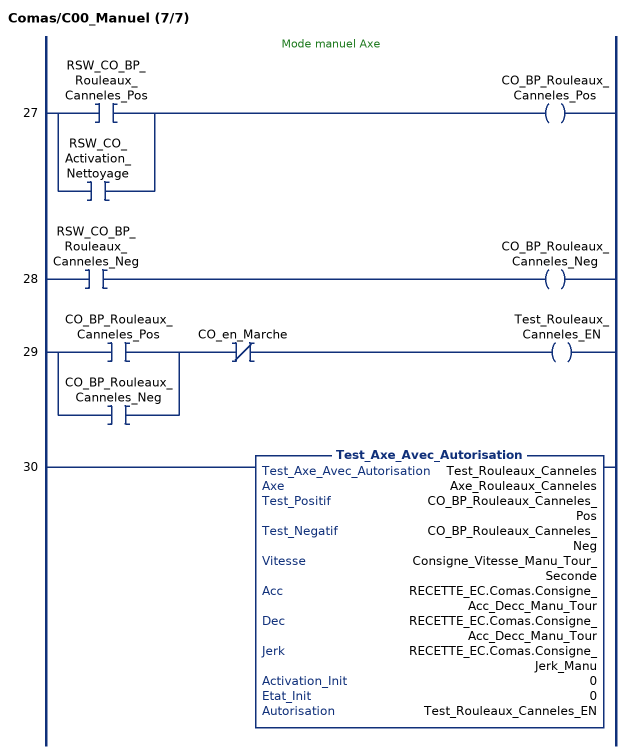
   // Mode manuel Axe
   27: [XIC(RSW_CO_BP_Rouleaux_Canneles_Pos) ,XIC(RSW_CO_Activation_Nettoyage) ]OTE(CO_BP_Rouleaux_Canneles_Pos);
   28: XIC(RSW_CO_BP_Rouleaux_Canneles_Neg)OTE(CO_BP_Rouleaux_Canneles_Neg);
   29: [XIC(CO_BP_Rouleaux_Canneles_Pos) ,XIC(CO_BP_Rouleaux_Canneles_Neg) ]XIO(CO_en_Marche)OTE(Test_Rouleaux_Canneles_EN);
   30: Test_Axe_Avec_Autorisation(Test_Rouleaux_Canneles,Axe_Rouleaux_Canneles,CO_BP_Rouleaux_Canneles_Pos,CO_BP_Rouleaux_Canneles_Neg,Consigne_Vitesse_Manu_Tour_Seconde,RECETTE_EC.Comas.Consigne_Acc_Decc_Manu_Tour,RECETTE_EC.Comas.Consigne_Acc_Decc_Manu_Tour,RECETTE_EC.Comas.Consigne_Jerk_Manu,0,0,Test_Rouleaux_Canneles_EN);
END_ROUTINE
